FUNCTION_BLOCK Timer EXTENDS Object
VAR_INPUT
END_VAR
VAR_OUTPUT
END_VAR
VAR
	_in: I_BoolSub;
	_q: I_BoolPub;
END_VAR

METHOD Refresh
VAR_INPUT
END_VAR
END_METHOD

END_FUNCTION_BLOCK

(* stored: Version 1.1.0.1, ProductVersion 3.1.4024.12
   POU Timer: Id {2a10577a-9a74-486a-885d-a513874d05e1}, SpecialFunc None
   Method Refresh: Id {59ff9bdd-5160-476b-9f55-fd8b157a0818} *)
